{attribute 'qualified_only'}
{attribute 'strict'}
TYPE E_Mode :
(
    Idle := 0,
    Running := 10,
    Done
) INT;
END_TYPE

(* stored: Version 1.1.0.1, ProductVersion 3.1.4024.12
   DUT E_Mode: Id {5f1c2d9e-0a6b-4c11-9d3e-7a1b2c3d4e21} *)
